Omron CX-Programmer project NewProject (CX-Programmer 9.73)

# PLC FACTORY_LAB: CP1H XA

## Program NewProgram1 (cyclic task 0)
Local symbols
Banda 100.00 BOOL
Etapa0 10.00 BOOL
Etapa1 10.01 BOOL
Etapa2 10.02 BOOL
Etapa3 10.03 BOOL
Etapa4 10.04 BOOL
Etapas 10 CHANNEL
Luz 100.01 BOOL
Sensor 0.02 BOOL
Start 0.00 BOOL
Stop 0.01 BOOL

### Section Section1

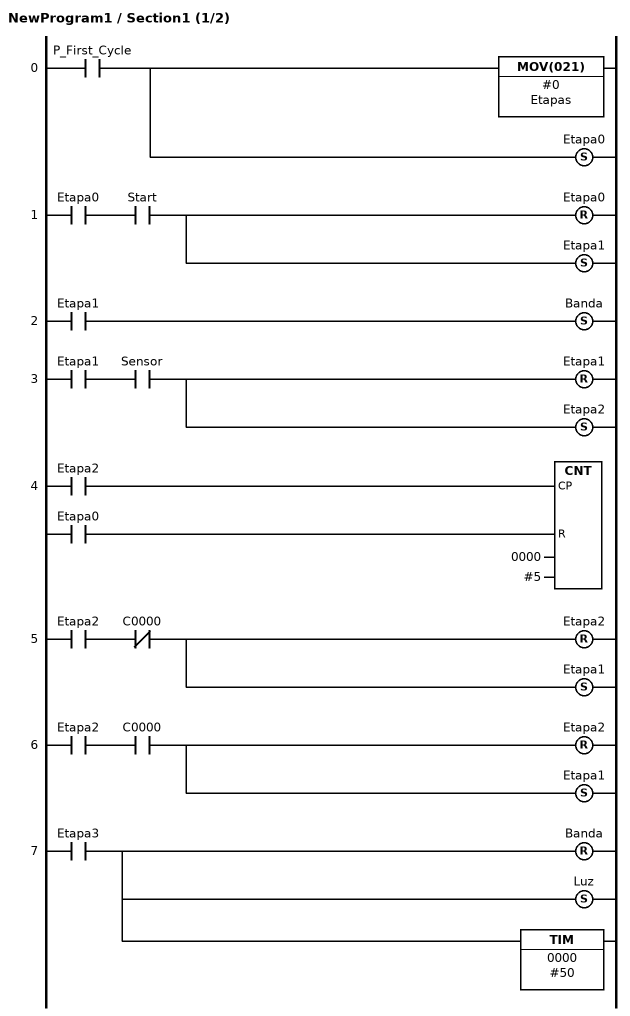
; rung 0
LD P_First_Cycle
MOV(021) #0 Etapas
SET Etapa0
; rung 1
LD Etapa0
AND Start
RSET Etapa0
SET Etapa1
; rung 2
LD Etapa1
SET Banda
; rung 3
LD Etapa1
AND Sensor
RSET Etapa1
SET Etapa2
; rung 4
LD Etapa2
LD Etapa0
CNT 0000 #5
; rung 5
LD Etapa2
ANDNOT C0000
RSET Etapa2
SET Etapa1
; rung 6
LD Etapa2
AND C0000
RSET Etapa2
SET Etapa1
; rung 7
LD Etapa3
RSET Banda
SET Luz
TIM 0000 #50

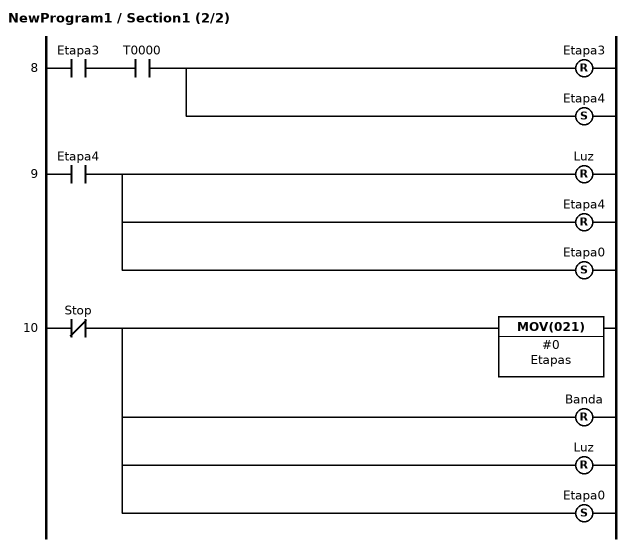
; rung 8
LD Etapa3
AND T0000
RSET Etapa3
SET Etapa4
; rung 9
LD Etapa4
RSET Luz
RSET Etapa4
SET Etapa0
; rung 10
LDNOT Stop
MOV(021) #0 Etapas
RSET Banda
RSET Luz
SET Etapa0

### Section END
; rung 0
END(001)